Yaskawa INFORM job: engine_planes_program.JBI

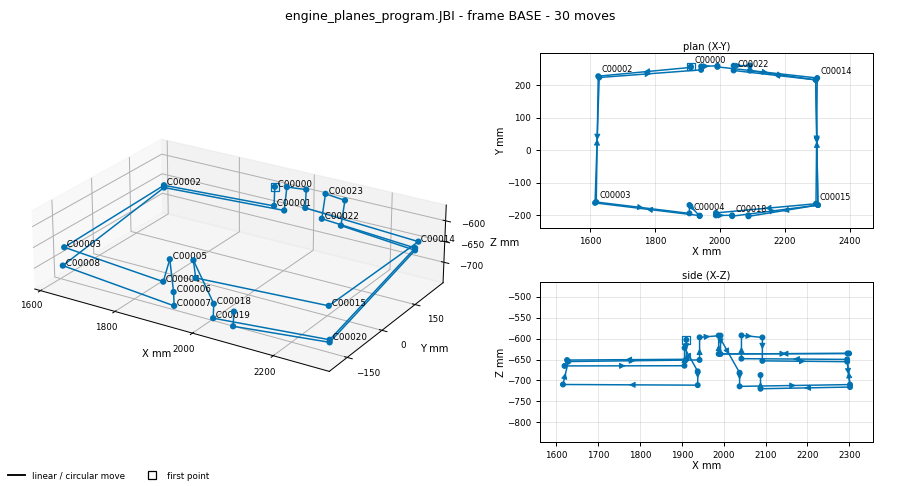
[picture p0: tool path of engine_planes_program.JBI in frame BASE, 30 of 32 moves have a stored position in this frame; points joined in program order, loops and branches not executed]
/JOB
//NAME engine_planes_program
//POS
///NPOS 30,0,30,0,0,0
///TOOL 0
///POSTYPE BASE
///RECTAN
///RCONF 0,0,0,0,0,0,0,0,0,0,0,0,0,0,0,0,0,0,0,0,0,0,0,0
C00000=1910.784114,258.264200,-603.105650,-175.000000,-5.000000,-5.000000
C00001=1910.756668,255.462505,-649.467881,175.000000,-43.714118,-90.561266
C00002=1625.907578,228.474214,-651.304212,141.523921,-23.655092,17.686406
C00003=1619.802959,-158.696297,-665.321723,175.000000,-46.003278,44.416205
C00004=1906.357025,-193.652475,-664.876011,175.000000,-46.285882,89.438734
C00005=1906.609407,-167.889352,-622.247624,175.000000,5.000000,5.000000
C00006=1938.003815,-201.791511,-678.207624,-175.000000,-5.000000,-5.000000
C00007=1938.016999,-200.445695,-711.294821,175.000000,-49.998465,89.438734
C00008=1616.130664,-161.395022,-709.686257,175.000000,-48.620446,44.023943
C00009=1628.934345,224.372385,-654.833796,144.585983,-23.365580,15.748054
C00010=1942.409249,247.914591,-651.025599,-175.000000,-40.001535,-90.561266
C00011=1942.515487,258.759390,-597.021624,175.000000,5.000000,5.000000
C00012=1992.532180,260.218508,-592.840624,-175.000000,-5.000000,-5.000000
C00013=1992.501361,257.072468,-636.769968,175.000000,-45.002365,-90.561266
C00014=2299.651787,222.870928,-635.511740,175.000000,-44.907363,-135.560943
C00015=2295.858217,-163.923401,-635.486543,-175.000000,-44.904116,134.438363
C00016=1988.101190,-192.096416,-636.741636,-175.000000,-44.997635,89.438734
C00017=1988.023966,-199.979411,-592.802624,175.000000,5.000000,5.000000
C00018=2038.030315,-199.576243,-681.500624,-175.000000,-5.000000,-5.000000
C00019=2038.004319,-202.229866,-714.156662,175.000000,-50.479061,89.438734
C00020=2301.786059,-168.097054,-709.891085,175.000000,-48.767155,134.990814
C00021=2295.066541,217.070221,-649.727483,145.567309,23.873548,-15.507021
C00022=2042.394975,245.967774,-648.002581,175.000000,-39.520939,-90.561266
C00023=2042.538950,260.664674,-592.383624,175.000000,5.000000,5.000000
C00024=2092.556875,261.228736,-597.340624,-175.000000,-5.000000,-5.000000
C00025=2092.401842,245.402966,-653.251545,-175.000000,-39.483726,-90.561266
C00026=2295.063672,217.025767,-655.226620,145.598378,23.870387,-15.488025
C00027=2301.855597,-168.118738,-715.806627,175.000000,-48.793361,134.998202
C00028=2088.011315,-202.781460,-719.862321,175.000000,-50.516274,89.438734
C00029=2088.045046,-199.338165,-687.141624,175.000000,5.000000,5.000000
///POSTYPE PULSE
///PULSE
EC00000=183296.0
EC00001=183296.0
EC00002=183296.0
EC00003=183296.0
EC00004=183296.0
EC00005=183296.0
EC00006=183296.0
EC00007=183296.0
EC00008=183296.0
EC00009=183296.0
EC00010=183296.0
EC00011=183296.0
EC00012=183296.0
EC00013=183296.0
EC00014=183296.0
EC00015=183296.0
EC00016=183296.0
EC00017=183296.0
EC00018=183296.0
EC00019=183296.0
EC00020=183296.0
EC00021=183296.0
EC00022=183296.0
EC00023=183296.0
EC00024=183296.0
EC00025=183296.0
EC00026=183296.0
EC00027=183296.0
EC00028=183296.0
EC00029=183296.0
//INST
///DATE 2023/08/16 18:17
///ATTR SC,RW,RJ
////FRAME BASE
///GROUP1 RB1,ST1
NOP
MOVJ P009 EX000 VJ=15.00
MOVJ C00000 EC00000 VJ=15.0
CALL JOB:SPYON
MOVL C00001 EC00001 V=150.0
MOVL C00002 EC00002 V=150.0
MOVL C00003 EC00003 V=150.0
MOVL C00004 EC00004 V=150.0
MOVL C00005 EC00005 V=150.0
MOVL C00006 EC00006 V=150.0
MOVL C00007 EC00007 V=150.0
MOVL C00008 EC00008 V=150.0
MOVL C00009 EC00009 V=150.0
MOVL C00010 EC00010 V=150.0
MOVL C00011 EC00011 V=150.0
MOVL C00012 EC00012 V=150.0
MOVL C00013 EC00013 V=150.0
MOVL C00014 EC00014 V=150.0
MOVL C00015 EC00015 V=150.0
MOVL C00016 EC00016 V=150.0
MOVL C00017 EC00017 V=150.0
MOVL C00018 EC00018 V=150.0
MOVL C00019 EC00019 V=150.0
MOVL C00020 EC00020 V=150.0
MOVL C00021 EC00021 V=150.0
MOVL C00022 EC00022 V=150.0
MOVL C00023 EC00023 V=150.0
MOVL C00024 EC00024 V=150.0
MOVL C00025 EC00025 V=150.0
MOVL C00026 EC00026 V=150.0
MOVL C00027 EC00027 V=150.0
MOVL C00028 EC00028 V=150.0
MOVL C00029 EC00029 V=150.0
CALL JOB:SPYOF
MOVJ P009 VJ=15.00
END
